# EPICS substitutions: kstar/siteApp/TS2/TS2App/Db/ts_value_B2.substitutions
#
file db/TS_CH_value.db
{
    pattern
        { DEV,    ID,       TAIL,     DESC,                ARG     }

        {"B2",    "0",      "VALUE",   "raw value",    "raw_cur"}
        {"B2",    "1",       "VALUE",   "raw value",    "raw_cur"}
        {"B2",    "2",       "VALUE",   "raw value",    "raw_cur"}
        {"B2",    "3",       "VALUE",   "raw value",    "raw_cur"}
        {"B2",    "4",       "VALUE",   "raw value",    "raw_cur"}
        {"B2",    "5",       "VALUE",   "raw value",    "raw_cur"}
        {"B2",    "6",       "VALUE",   "raw value",    "raw_cur"}
        {"B2",    "7",       "VALUE",   "raw value",    "raw_cur"}
        {"B2",    "8",       "VALUE",   "raw value",    "raw_cur"}
        {"B2",    "9",       "VALUE",   "raw value",    "raw_cur"}
        {"B2",    "10",       "VALUE",   "raw value",    "raw_cur"}
        {"B2",    "11",       "VALUE",   "raw value",    "raw_cur"}
        {"B2",    "12",       "VALUE",   "raw value",    "raw_cur"}
        {"B2",    "13",       "VALUE",   "raw value",    "raw_cur"}
        {"B2",    "14",       "VALUE",   "raw value",    "raw_cur"}
        {"B2",    "15",       "VALUE",   "raw value",    "raw_cur"}

}
